// TwinCAT 3 PLC project TestHMI
// ProgramVersion: 3.1.4024.0
// libraries:
//   Tc2_Standard, * (Beckhoff Automation GmbH)
//   Tc2_System, * (Beckhoff Automation GmbH)
//   Tc3_Module, * (Beckhoff Automation GmbH)
//   VisuDialogs, * (System)
// project tree:
//   / GlobalTextList.TcGTLO, TestHMI.TcTTO, 视图管理器.TcVMO (not stored)
//   POUs/ MAIN.TcPOU
//   VISUs/ AxisGroupStateList.TcTLO, MainStateList.TcTLO, SafetyStatusList.TcTLO, SpindleStateList.TcTLO, TestHMI.TcVIS
// (motion and I/O tree: see PLC project portal)
// real-time tasks:
//   TASK PlcTask: cycle T#250us, priority 10, ADS port 350
//   TASK MotionControl: cycle T#250us, priority 4, ADS port 352
//   TASK ModuleSpindle: cycle T#250us, priority 6, ADS port 351
//   TASK ModuleAxisGroup: cycle T#250us, priority 8, ADS port 353
//   TASK ModuleTest: cycle T#250us, priority 12, ADS port 354
//   TASK TestHMI: cycle T#10ms, priority 18, ADS port 355
//   TASK ModuleSafety: cycle T#250us, priority 14, ADS port 356
// variable links:

CONFIGURATION TestHMI
    RESOURCE PLC ON TwinCAT3
        TASK TestHMI(INTERVAL := T#10ms, PRIORITY := 18);
        PROGRAM MAIN WITH TestHMI : MAIN;
    END_RESOURCE
END_CONFIGURATION

// ---- POUs/MAIN.TcPOU
PROGRAM MAIN
VAR
	MockPanel AT%Q*: PanelInfo;
	Recovery AT%Q*: BOOL;
	ContinuousMoving AT%Q*: BOOL;
	
	SpindleCW : BOOL;
	SpindleCCW : BOOL;
	
	Axis_X : BOOL;
	Axis_Y : BOOL;
	Axis_Z : BOOL;
	IncrementalPos : INT;
	Ratio_01 : BOOL;
	Ratio_001 : BOOL;
	Ratio_0001 : BOOL;
	
	TestAxisGroupState AT%I*: AxisGroupState;
	TestSpindleState AT%I*: SpindleState;
	AxisGroupStateListId : INT;
	SpindleStateListId : INT;
	
	TestMainState AT%I*: SystemState;
	TestSafetyStatus AT%I*: SafetyState;
	MainStateListId : INT;
	SafetyStatusListId : INT;
END_VAR

IF SpindleCW THEN
	MockPanel.Spindle_Cmd := 1;
ELSIF SpindleCCW THEN
	MockPanel.Spindle_Cmd := -1;
ELSE
	MockPanel.Spindle_Cmd := 0;
END_IF

IF Ratio_01 THEN
	MockPanel.Handwheel_Ratio := 0.1;
ELSIF Ratio_001 THEN
	MockPanel.Handwheel_Ratio := 0.01;
ELSIF Ratio_0001 THEN
	MockPanel.Handwheel_Ratio := 0.001;
ELSE
	MockPanel.Handwheel_Ratio := 1.0;
END_IF

IF Axis_X THEN
	MockPanel.Handwheel_EnabledAxisNum := AxisOrder.Axis_X;
	MockPanel.Handwheel_dPos[0] := INT_TO_LREAL(IncrementalPos) * MockPanel.Handwheel_Ratio;
ELSIF Axis_Y THEN
	MockPanel.Handwheel_EnabledAxisNum := AxisOrder.Axis_Y;
	MockPanel.Handwheel_dPos[1] := INT_TO_LREAL(IncrementalPos) * MockPanel.Handwheel_Ratio;
ELSIF Axis_Z THEN
	MockPanel.Handwheel_EnabledAxisNum := AxisOrder.Axis_Z;
	MockPanel.Handwheel_dPos[2] := INT_TO_LREAL(IncrementalPos) * MockPanel.Handwheel_Ratio;
ELSE
	MockPanel.Handwheel_EnabledAxisNum := 0;
END_IF

AxisGroupStateListId := TO_INT(TestAxisGroupState);
SpindleStateListId := TO_INT(TestSpindleState);
MainStateListId := TO_INT(TestMainState);
SafetyStatusListId := TO_INT(TestSafetyStatus);

END_PROGRAM

// ---- GlobalTextList.TcGTLO
TEXTLIST GlobalTextList
  972 = '%s'
  178 = '0.001'
  243 = '0.01'
  489 = '0.1'
  845 = 'COntinuousMOving'
  62 = 'COntinuousMoving'
  223 = 'ContinuousMoving'
  108 = 'Recovery'
  517 = 'Reset'
  381 = 'Servo'
  417 = 'Spindle CCW'
  353 = 'Spindle CW'
  762 = 'Spindle Stop'
  83 = 'X'
  644 = 'Y'
  698 = 'Z'
END_TEXTLIST

// ---- VISUs/AxisGroupStateList.TcTLO
TEXTLIST AxisGroupStateList
  0 = 'AxisGroupIdle'
  1 = 'AxisGroupInitialization'
  2 = 'AxisGroupDisabled'
  3 = 'AxisGroupPreStandby'
  4 = 'AxisGroupStandby'
  5 = 'AxisGroupManualMoving'
  6 = 'AxisGroupPreContinuousMoving'
  7 = 'AxisGroupContinuousMoving'
  8 = 'AxisGroupLimitViolation'
  9 = 'AxisGroupEmergency'
  10 = 'AxisGroupFault'
  11 = 'AxisGroupRecovery'
  13 = 'AxisGroupPositioning'
   = ''
END_TEXTLIST

// ---- VISUs/MainStateList.TcTLO
TEXTLIST MainStateList
  0 = 'Idle'
  1 = 'Disabled'
  2 = 'PreStandby'
  3 = 'Standby'
  4 = 'Manual'
  5 = 'Buffering'
  6 = 'ContinuousExecution'
  7 = 'Fault'
  8 = 'Test'
  9 = 'Recovery'
   = ''
END_TEXTLIST

// ---- VISUs/SafetyStatusList.TcTLO
TEXTLIST SafetyStatusList
  0 = 'SafetyStateNormal'
  1 = 'SafetyStateWarning'
  2 = 'SafetyStateEmergency'
  3 = 'SafetyStateFault'
  4 = 'SafetyStateRecovery'
   = ''
END_TEXTLIST

// ---- VISUs/SpindleStateList.TcTLO
TEXTLIST SpindleStateList
  0 = 'SpindleIdle'
  1 = 'SpindleInitialization'
  2 = 'SpindleDisabled'
  3 = 'SpindleEnable'
  4 = 'SpindlePreMoving'
  5 = 'SpindleRotating'
  6 = 'SpindlePositioning'
  7 = 'SpindlePostMoving'
  8 = 'SpindleEmergency'
  9 = 'SpindleFault'
  10 = ''
   = ''
END_TEXTLIST

// ---- VISUs/TestHMI.TcVIS
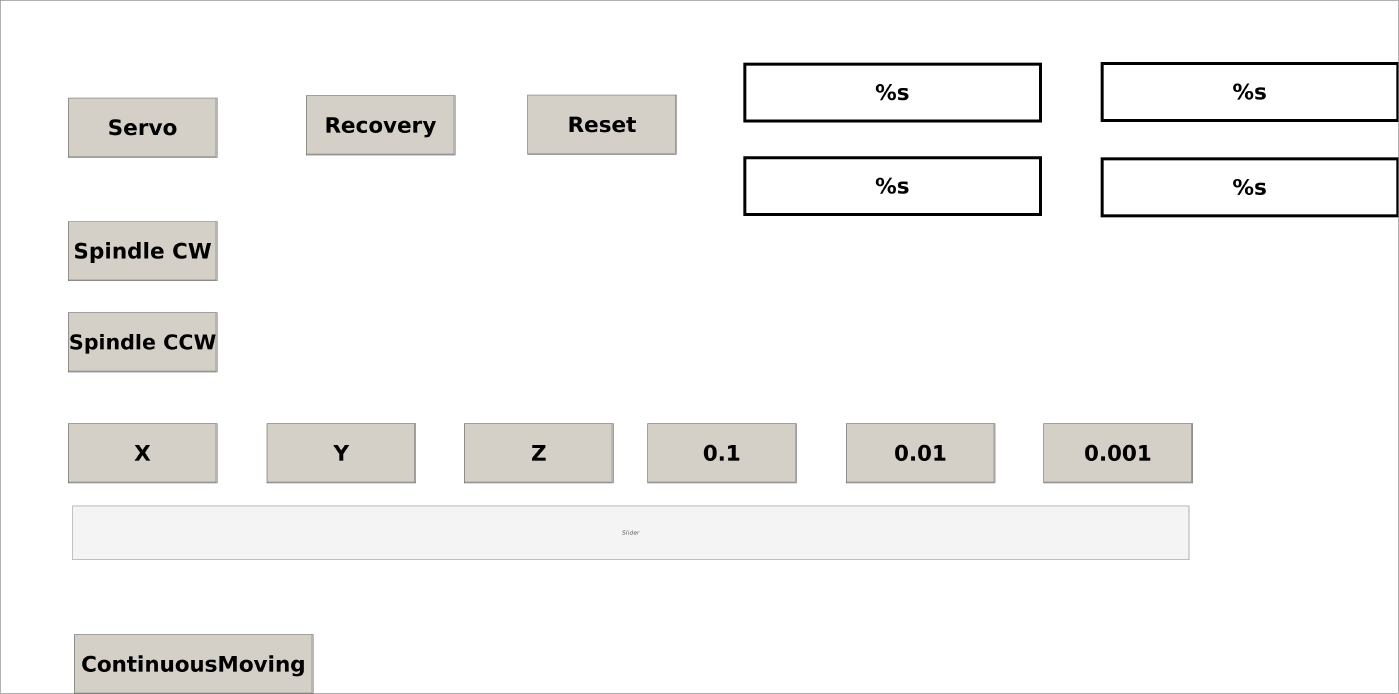
VISUALIZATION TestHMI  // 2345x1164
    Button (114,164 250x100), "Servo", colour toggle: MAIN.MockPanel.ServoOn
        toggle MAIN.MockPanel.ServoOn
    Button (114,371 250x100), "Spindle CW", colour toggle: MAIN.SpindleCW, input disabled if: MAIN.SpindleCCW
        toggle MAIN.SpindleCW
    Button (114,524 250x100), "Spindle CCW", colour toggle: MAIN.SpindleCCW, input disabled if: MAIN.SpindleCW
        toggle MAIN.SpindleCCW
    Slider (121,848 1872x91), variable: MAIN.IncrementalPos, scale -20..20
    Button (114,710 250x100), "X", colour toggle: MAIN.Axis_X
        toggle MAIN.Axis_X
        OnMouseDown: execute { MAIN.MockPanel.Handwheel_EnabledAxisNum := 1; }
    Button (447,710 250x100), "Y", colour toggle: MAIN.Axis_Y
        toggle MAIN.Axis_Y
        OnMouseDown: execute { MAIN.MockPanel.Handwheel_EnabledAxisNum := 2; }
    Button (778,710 250x100), "Z", colour toggle: MAIN.Axis_Z
        toggle MAIN.Axis_Z
        OnMouseDown: execute { MAIN.MockPanel.Handwheel_EnabledAxisNum := 3; }
    Rectangle (1246,105 500x100), "%s", text list: 'AxisGroupStateList', text index: MAIN.AxisGroupStateListId
    Rectangle (1246,262 500x100), "%s", text list: 'SpindleStateList', text index: MAIN.SpindleStateListId
    Button (1085,710 250x100), "0.1", colour toggle: MAIN.Ratio_01
        toggle MAIN.Ratio_01
        OnMouseDown: execute { MAIN.MockPanel.Handwheel_EnabledAxisNum := 1; }
    Button (1418,710 250x100), "0.01", colour toggle: MAIN.Ratio_001
        toggle MAIN.Ratio_001
        OnMouseDown: execute { MAIN.MockPanel.Handwheel_EnabledAxisNum := 2; }
    Button (1749,710 250x100), "0.001", colour toggle: MAIN.Ratio_0001
        toggle MAIN.Ratio_0001
        OnMouseDown: execute { MAIN.MockPanel.Handwheel_EnabledAxisNum := 3; }
    Rectangle (1845,104 500x100), "%s", text list: 'MainStateList', text index: MAIN.MainStateListId
    Rectangle (1845,264 500x100), "%s", text list: 'SafetyStatusList', text index: MAIN.SafetyStatusListId
    Button (513,160 250x100), "Recovery", colour toggle: MAIN.Recovery
        toggle MAIN.Recovery
    Button (884,159 250x100), "Reset", colour toggle: MAIN.MockPanel.Reset
        toggle MAIN.MockPanel.Reset
    Button (124,1064 401x100), "ContinuousMoving", colour toggle: MAIN.ContinuousMoving
        toggle MAIN.ContinuousMoving
        OnMouseDown: execute { MAIN.MockPanel.Handwheel_EnabledAxisNum := 1; }
END_VISUALIZATION
